FUNCTION_BLOCK Blinker
VAR_INPUT
	bStartBlinker : BOOL; //bool variable that starts the blinker
END_VAR
VAR_OUTPUT
	bStatus : BOOL; //bool variable that transfers the blinkers output status to the light
END_VAR
VAR
	fbTimer1 : TON; //timers for every on/off state
	fbTimer2 : TON;
	fbTimer3 : TON;
END_VAR

IF bStartBlinker THEN // if the blinker starts execute
	
fbTimer2.IN := TRUE; //starts the time
	IF fbTimer2.Q THEN
		bStatus := FALSE; //sets the light to off
		fbTimer1.IN := TRUE; //starts the new timer
	END_IF

	IF fbTimer1.Q THEN
		bStatus := TRUE; //sets the light to on
		fbTimer3.IN := TRUE; //turns the reset timer
	END_IF
	
	IF fbTimer3.Q THEN
		fbTimer1.IN := FALSE; //resets all the timers
		fbTimer2.IN := FALSE;
		fbTimer3.IN := FALSE;
	END_IF
END_IF
fbTimer1(PT := T#15MS); //timers for the on/off states
fbTimer2(PT := T#15MS);
fbTimer3(PT := T#15MS);

END_FUNCTION_BLOCK

(* stored: Version 1.1.0.1, ProductVersion 3.1.4024.12
   POU Blinker: Id {8e5b29d9-5298-4e40-af5f-a7868ce84bdc}, SpecialFunc None *)
